
FUNCTION CB_gt_tod : BOOL


TITLE = ' Test Whether IN0 is strictly greater than IN1 '
VERSION : '1.0'
AUTHOR  : CB
NAME    : gt_tod
FAMILY  : TNI

VAR_INPUT
    IN0 : TOD;
    IN1 : TOD;
END_VAR

BEGIN

CB_gt_tod := (IN0 > IN1);

END_FUNCTION
